FUNCTION_BLOCK FB_FixedMotor IMPLEMENTS I_Motor

VAR
	bRunning : BOOL;
END_VAR

{warning 'add method implementation '}
METHOD Start : BOOL
bRunning := TRUE;
Start := bRunning;
END_METHOD

{warning 'add method implementation '}
METHOD Stop : BOOL
bRunning := FALSE;
Stop := NOT bRunning;
END_METHOD

END_FUNCTION_BLOCK

(* stored: Version 1.1.0.1, ProductVersion 3.1.4024.16
   POU FB_FixedMotor: Id {793e6d71-4619-4cbf-a568-8200bbbdbf3f}, SpecialFunc None
   Method Start: Id {71f5b658-6d4b-4388-81cd-cc22acf28875}
   Method Stop: Id {d95b4897-9ea5-4781-b578-ffadc6797259} *)
